TYPE NewtonMeter : LREAL;
END_TYPE

(* stored: Version 1.1.0.1, ProductVersion 3.1.4024.12
   DUT NewtonMeter: Id {37e06295-d7dd-46ae-961a-b5aca1322381} *)
